// TIA Portal V18 export
DATA_BLOCK "HMISystemDB"   // DB2201
{ S7_Optimized_Access := 'FALSE' }
VERSION : 0.1
// stored: AutoNumber false, DBAccessibleFromOPCUA true, DBAccessibleFromWebserver true, IsOnlyStoredInLoadMemory false, IsWriteProtectedInAS false
   VAR RETAIN
      DisplayRows : Int;
      MaxPage : Int;
      Rows : Int;
      UnEnableGroup : Bool;
      DisplaySymbol : Bool;
      "DisplaySymbol Time" : Int;
      SymbolText : Array[1..4] of Int;
      HMICylinderBypass : Array[1..50] of Struct
         "BY" : Array[1..50] of Int;
      END_STRUCT;
      HMI_Axis : "HMI_Axis";
   END_VAR
BEGIN
   HMI_Axis.INPUT.Axis_ID := 1;
END_DATA_BLOCK
